Staubli VAL3: onF2Event.pgx

program onF2Event()
begin
end
